// TIA Portal V20 export
TYPE "typeEnMeterRestore"
TITLE = Energy Meter Restore / Energy meter restore
// Struktur Energy Meter Restore / Structure energy meter restore
// stored: Access Published
   STRUCT
      dataRecordVersion : Byte;   // dataRecordVersion
      reserved : Byte;   // Reserve / Reserved
      controlByte1L1 : Byte;   // Control byte1 L1
      controlByte2L1 : Byte;   // Control byte2 L1
      controlByte1L2 : Byte;   // Control byte1 L2
      controlByte2L2 : Byte;   // Control byte2 L2
      controlByte1L3 : Byte;   // Control byte1 L3
      controlByte2L3 : Byte;   // Control byte2 L3
      effEnImportL1 : LReal;   // Energie Wirkleistung Import L1 / Effective energy import L1
      effEnExportL1 : LReal;   // Energie Wirkleistung Export L1 / Effective energy export L1
      reaEnImportL1 : LReal;   // Energie Blindleistung Import L1 / Reactive energy import L1
      reaEnExportL1 : LReal;   // Energie Blindleistung Export L1 / Reactive energy export L1
      appEnL1 : LReal;   // Energie Scheinleistung L1 / Apparent energy L1
      effEnImportL2 : LReal;   // Energie Wirkleistung Import L2 / Effective energy import L2
      effEnExportL2 : LReal;   // Energie Wirkleistung Export L2 / Effective energy export L2
      reaEnImportL2 : LReal;   // Energie Blindleistung Import L2 / Reactive energy import L2
      reaEnExportL2 : LReal;   // Energie Blindleistung Export L2 / Reactive energy export L2
      appEnL2 : LReal;   // Energie Scheinleistung L2 / Apparent energy L2
      effEnImportL3 : LReal;   // Energie Wirkleistung Import L3 / Effective energy import L3
      effEnExportL3 : LReal;   // Energie Wirkleistung Export L3 / Effective energy export L3
      reaEnImportL3 : LReal;   // Energie Blindleistung Import L3 / Reactive energy import L3
      reaEnExportL3 : LReal;   // Energie Blindleistung Export L3 / Reactive energy export L3
      appEnL3 : LReal;   // Energie Scheinleistung L3 / Apparent energy L3
   END_STRUCT;
END_TYPE
